KUKA KRL program: AprilTag.src, AprilTag.dat

--- AprilTag.src ---
&ACCESS RVP
&PARAM EDITMASK = *
DEF AprilTag()
   ; AprilTagExample
   ; --------------
   ; Demonstrates AprilTag detection and robot positioning using Roboception's AprilTag module. The program:
   ; 1. Configures detection parameters
   ; 2. Performs AprilTag detection
   ; 3. For each detected tag, moves robot to corresponding positions
   ; 4. Returns to home position after completion
   ;

   ; Service name - same as the EKI service name
   ; TODO: Change this to the correct service name - could be "rc_april_tag_detect-detect"
   serviceNameDetect[] = "rc_april_tag_detect-detect"

   ; Initialize robot and set up interrupts
   ;FOLD INI;%{PE}
      ;FOLD BASISTECH INI
         GLOBAL INTERRUPT DECL 3 WHEN $STOPMESS==TRUE DO IR_STOPM ( )
         INTERRUPT ON 3
         BAS (#INITMOV,0 )
      ;ENDFOLD (BASISTECH INI)
   ;ENDFOLD (INI)

   ; Initialize message received interrupt for EKI communication
   INTERRUPT DECL 89 WHEN $FLAG[998] DO RC_NOTIFYRECEIVED(1, 998)
   INTERRUPT ON 89

   ; Move robot to home position
   MoveToStartPosition()

   ; Initialize AprilTag detection and open connection to rc_cube
   $FLAG[1] = FALSE
   RC_SETMSG("Starting AprilTag detection")

   RC_INIT(serviceNameDetect[])

   ; Configure and perform detection
   ConfigureDetection(serviceNameDetect[])
   PerformDetection(serviceNameDetect[])

   ; Process results
   IF DetectionSuccessful() THEN
      ExecuteTagMovements()
   ELSE
      HandleDetectionFailure()
   ENDIF

   ; Cleanup
   RC_SETMSG("Detection finished")

   ; Return to home position
   MoveToStartPosition()
END

DEF ExecuteTagMovements()
   DECL INT i
   DECL FRAME AprilPose

   FOR i=1 TO NUMDETECTEDTAGS
      AprilPose = DETECTEDTAGS[i]
      MoveToTagPosition(AprilPose)
   ENDFOR
END

DEF MoveToTagPosition(AprilPose:IN)
   DECL FRAME AprilPose
   DECL FRAME AboveAprilPose
   AboveAprilPose = AprilPose
   AboveAprilPose.Z = AprilPose.Z + 100

   SPTP AboveAprilPose WITH $VEL_AXIS[1] = SVEL_JOINT(100.0), $TOOL = STOOL2(FP1), $BASE = SBASE(FP1.BASE_NO), $IPO_MODE = SIPO_MODE(FP1.IPO_FRAME), $LOAD = SLOAD(FP1.TOOL_NO), $ACC_AXIS[1] = SACC_JOINT(PPDAT1), $APO = SAPO_PTP(PPDAT1), $GEAR_JERK[1] = SGEAR_JERK(PPDAT1), $COLLMON_TOL_PRO[1] = USE_CM_PRO_VALUES(0)
END

DEF MoveToStartPosition()
   ;FOLD SPTP STARTPOSE Vel=100 % DEFAULT
      SPTP STARTPOSE WITH $VEL_AXIS[1]= SVEL_JOINT(100), $TOOL= STOOL2(fDatDefault), $BASE= SBASE(fDatDefault.BASE_NO), $IPO_MODE= SIPO_MODE(fDatDefault.IPO_FRAME), $LOAD= SLOAD(fDatDefault.TOOL_NO), $ACC_AXIS[1]= SACC_JOINT(PDEFAULT), $GEAR_JERK[1]= SGEAR_JERK(PDEFAULT)
   ;ENDFOLD
END


; ---- Roboception Functions ----
;FOLD RC Functions
   DEF ConfigureDetection(serviceNameDetect[]:IN)
      ; Configures detection parameters for AprilTag detection
      ;
      ; @param serviceNameDetect[]: EKI configuration/service name
      ;
      DECL CHAR serviceNameDetect[]
      DECL EKI_Status RET
      DECL E6POS flangePose

      flangePose = $POS_ACT_MES : INV_POS($TOOL)

      RET = EKI_SetString(serviceNameDetect[], "req/args/pose_frame", "external")
      RET = EKI_SetFrame(serviceNameDetect[], "req/args/robot_pose", flangePose)
   END

   DEF PerformDetection(serviceNameDetect[]:IN)
      ; Performs AprilTag detection using configured parameters
      ;
      ; @param serviceNameDetect[]: EKI configuration/service name
      ;
      DECL CHAR serviceNameDetect[]
      DECL EKI_Status RET

      ; Open connection before sending request
      RC_OPENCONNECTION(serviceNameDetect[])

      ; Synchronize advance run pointer
      WAIT SEC 0

      ; Send request
      RET = EKI_Send(serviceNameDetect[], "req")

      ; Wait for response and read results
      RC_WAITFORRESULT(1)
      RC_READRESULT(serviceNameDetect[])

      ; Close the connection after reading results
      RC_CLOSECONNECTION(serviceNameDetect[], "req")
   END

   DEFFCT BOOL DetectionSuccessful()
      ; Checks if AprilTag detection was successful
      ;
      ; @return TRUE if tags were detected, FALSE otherwise
      ;
      IF(RETURNCODE.VALUE < 0) THEN
         RETURN FALSE
      ENDIF

      IF NUMDETECTEDTAGS > 0 THEN
         ShowDetectionResults()
         RETURN TRUE
      ENDIF

      RETURN FALSE
   ENDFCT

   DEF ShowDetectionResults()
      ; Displays information about detected AprilTags
      ;
      DECL INT i
      DECL KrlMsgPar_T countPar[1]
      DECL KrlMsgPar_T par[4]

      countPar[1] = {par_type #value, par_real 0}
      countPar[1].par_real = NUMDETECTEDTAGS
      RC_SETMSG_PARAM("Number of AprilTags detected: %1", countPar[])

      FOR i=1 TO NUMDETECTEDTAGS
         par[1] = {par_type #value, par_real 0}
         par[1].par_real = i
         par[2] = {par_type #value, par_real 0}
         par[2].par_real = DETECTEDTAGS[i].X
         par[3] = {par_type #value, par_real 0}
         par[3].par_real = DETECTEDTAGS[i].Y
         par[4] = {par_type #value, par_real 0}
         par[4].par_real = DETECTEDTAGS[i].Z
         RC_SETMSG_PARAM("April Tag %1: X: %2, Y: %3, Z: %4", par[])
      ENDFOR
   END

   DEF HandleDetectionFailure()
      ; Handles cases where AprilTag detection fails
      ;
      IF(RETURNCODE.VALUE < 0) THEN
         RC_SETMSG("Execution failed")
      ELSE
         RC_SETMSG("No AprilTags detected")
      ENDIF
   END

   DEF RC_SETMSG(msg[]:IN)
      DECL CHAR msg[]
      DECL KrlMsgPar_T params[3]

      RC_SETMSG_PARAM(msg[], params[])
   END

   DEF RC_SETMSG_PARAM(msg[]:IN, params[]:OUT)
      DECL CHAR msg[]
      DECL KrlMsgPar_T params[]

      DECL KrlMsg_T name
      DECL KrlMsgOpt_T options
      DECL INT Handle, len, count
      DECL EKrlMsgType Type

      name={modul[] "rc", nr 1, msg_txt[] " "}
      Type=#notify

      len=STRLEN(msg[])
      IF len>0 THEN
         IF len>80 THEN
            len=80
         ENDIF
         FOR count=1 TO len
            name.msg_txt[count]=msg[count]
         ENDFOR
      ELSE
         name.msg_txt[]="parameter msg[] is missing"
      ENDIF

      Handle=Set_KrlMsg(Type, name, params[], options)
   END

   DEF RC_INIT(configFileName[]:IN)
      DECL CHAR configFileName[]
      DECL EKI_Status RET
      RET=EKI_INIT(configFileName[])
   END

   DEF RC_OPENCONNECTION(configFileName[]:IN)
      DECL CHAR configFileName[]
      DECL EKI_Status RET
      RET=EKI_Open(configFileName[])
      EKI_CHECK(RET,#Quit)
   END

   DEF RC_CLOSECONNECTION(configFileName[]:IN, strPlace[]:IN)
      DECL CHAR configFileName[]
      DECL CHAR strPlace[]
      DECL EKI_Status RET
      WAIT SEC 0
      RET=EKI_Close(configFileName[])
      RET=EKI_ClearBuffer(configFileName[], strPlace[])
   END

   DEF RC_WAITFORRESULT(WaitFlag:IN)
      DECL INT WaitFlag
      WAIT FOR $FLAG[WaitFlag] OR NOT $FLAG[RCEkiAliveFlagNo]
      IF(NOT $FLAG[RCEkiAliveFlagNo]) THEN
         RC_SETMSG("EKI connection lost")
      ENDIF
      $FLAG[WaitFlag] = FALSE
      WAIT SEC 0
   END

   DEF RC_NOTIFYRECEIVED(WAITFLAG:IN, EOFRESULFLAG:IN)
      DECL INT WAITFLAG
      DECL INT EOFRESULFLAG
      $FLAG[EOFRESULFLAG]=FALSE
      $FLAG[WAITFLAG]=TRUE
   END

   DEF RC_READRESULT(configFileName[]:IN)
      DECL CHAR configFileName[]
      DECL RETURNCODE_T RESULT
      DECL EKI_STATUS RET
      DECL INT j
      DECL FRAME POSE

      POSE = POSE_IDENT
      RESULT={VALUE 0, MSG[] "0"}

      RET = EKI_GetInt(configFileName[], "res/return_code/@value", RESULT.VALUE)
      RET = EKI_GetString(configFileName[], "res/return_code/@message", RESULT.MSG[])
      RETURNCODE = RESULT

      ; Display error message immediately if there is one
      IF (RESULT.VALUE < 0) THEN
         RC_SETMSG("API Error")
         RC_SETMSG(RESULT.MSG[])
      ENDIF

      RET = EKI_CheckBuffer(configFileName[], "res/tags/le/id")
      NUMDETECTEDTAGS = RET.Buff

      FOR j=1 TO NUMDETECTEDTAGS
         RET = EKI_GetFrame(configFileName[], "res/tags/le/pose", POSE)
         DETECTEDTAGS[j] = POSE
      ENDFOR

      RET = EKI_ClearBuffer(configFileName[], "res")
   END
;ENDFOLD (RC Functions)

--- AprilTag.dat ---
&ACCESS RVP
&PARAM EDITMASK = *
DEFDAT AprilTag

   ;FOLD EXTERNAL DECLARATIONS;%{PE}%MKUKATPBASIS,%CEXT,%VCOMMON,%P
   ;FOLD BASISTECH EXT;%{PE}%MKUKATPBASIS,%CEXT,%VEXT,%P
   EXT  BAS (BAS_COMMAND  :IN,REAL  :IN )
   ;ENDFOLD (BASISTECH EXT)
   ;FOLD USER EXT;%{E}%MKUKATPUSER,%CEXT,%VEXT,%P
   ;Make your modifications here

   ; Common structures and variables
   STRUC RETURNCODE_T INT VALUE,CHAR MSG[512]
   DECL INT RCEkiAliveFlagNo=997
   DECL RETURNCODE_T RETURNCODE
   DECL FRAME POSE_IDENT={X 0.0,Y 0.0,Z 0.0,A 0.0,B 0.0,C 0.0}

   ; Service configuration
   DECL CHAR serviceNameDetect[64]

   ; Detection results
   DECL FRAME DETECTEDTAGS[32]
   DECL INT NUMDETECTEDTAGS

   ; Frame data
   DECL FDAT FP1={TOOL_NO 4,BASE_NO 0,IPO_FRAME #BASE,POINT2[] " "}

   ; Point data
   DECL PDAT PPDAT1={VEL 100.0,ACC 100.0,APO_DIST 100.0,APO_MODE #CPTP,GEAR_JERK 50.0,EXAX_IGN 0}

   ; Start position
   DECL E6POS STARTPOSE={X 0,Y 0,Z 0,A 0,B 0,C 0,S 0,T 0,E1 0.0,E2 0.0,E3 0.0,E4 0.0,E5 0.0,E6 0.0}

   ; Movement data
   DECL LDAT lDatDefault={VEL 2.00000,ACC 20.0000,APO_DIST 10.0000,APO_FAC 50.0000,AXIS_VEL 100.000,AXIS_ACC 100.000,ORI_TYP #VAR,CIRC_TYP #BASE,JERK_FAC 50.0000,GEAR_JERK 100.000,EXAX_IGN 0,CB {AUX_PT {ORI #CONSIDER,E1 #CONSIDER,E2 #CONSIDER,E3 #CONSIDER,E4 #CONSIDER,E5 #CONSIDER,E6 #CONSIDER},TARGET_PT {ORI #INTERPOLATE,E1 #INTERPOLATE,E2 #INTERPOLATE,E3 #INTERPOLATE,E4 #INTERPOLATE,E5 #INTERPOLATE,E6 #INTERPOLATE}}}
   DECL FDAT fDatDefault={TOOL_NO 4,BASE_NO 0,IPO_FRAME #BASE,POINT2[] " "}
   DECL PDAT pDatDefault={VEL 10.0000,ACC 20.0000,APO_DIST 10.0000,APO_MODE #CDIS,GEAR_JERK 100.000,EXAX_IGN 0}

   ;ENDFOLD (USER EXT)
   ;ENDFOLD (EXTERNAL DECLARATIONS)
ENDDAT
